Staubli VAL3: page_Template4.pjx

--- page_Template4.pjx ---
Parameters version=s7.7.1 stackSize=5000 millimeterUnit=true
Program file=buildList.pgx
Program file=listAdd.pgx
Program file=loadPage.pgx
Program file=main.pgx
Program file=onEnterEvent.pgx
Program file=onExit.pgx
Program file=onF1Event.pgx
Program file=onF2Event.pgx
Program file=onF3Event.pgx
Program file=onF4Event.pgx
Program file=onF5Event.pgx
Program file=onF6Event.pgx
Program file=onF7Event.pgx
Program file=onF8Event.pgx
Program file=onStart.pgx
Program file=refresh.pgx
Program file=refreshDynamic.pgx
Program file=refreshStatic.pgx
Data file=page_Template4.dtx
Library alias=page path=Disk://kernel/template/page/page.pjx
Library alias=use path=Disk://kernel/userPage/userPage.pjx
Library alias=language path=Disk://kernel/language/language.pjx
Library alias=global path=Disk://saveData/saveData.pjx

--- loadPage.pgx ---
program loadPage(string x_sPage, string& x_sItems[])
// load the next page
  local num i
begin
  // look if the page libload is correct
  i=page:libLoad(x_sPage)
  if i!=0
    logMsg("[VALPLAST] INTERFACE:PAGE LIBLOAD "+x_sPage+" result "+toString("",i))
    popUpMsg("Loading page "+x_sPage+" error CODE "+toString("",i))
  else
    // copy all the field from x_sItems to the next page
    call use:stringCopy(x_sItems,page:sItems)
    call page:main()
    // to give back
    call use:stringCopy(page:sItems,x_sItems)
  endIf
end

--- onEnterEvent.pgx ---
program onEnterEvent()
begin
  //
  // NB sEvent is the selected
  // element in the LIST
  //
end

--- onF3Event.pgx ---
program onF3Event()
begin
  // look if the bButton is enable
  if bButton[2]
    //
  endIf
end

--- onF6Event.pgx ---
program onF6Event()
begin
   // look if the bButton is enable
  if bButton[5]
    //
  endIf
    end

--- onF7Event.pgx ---
program onF7Event()
begin
   // look if the bButton is enable
  if bButton[6]
    //
  endIf
   end

--- onF8Event.pgx ---
program onF8Event()
begin
   // look if the bButton is enable
  if bButton[7]
    //
  endIf
end

--- refreshDynamic.pgx ---
program refreshDynamic()
begin
  // DO NOT CHANGE
  nRefresh=clock()
  use:bUseRefresh=false
  //
  // ADD HERE
  //
 end
